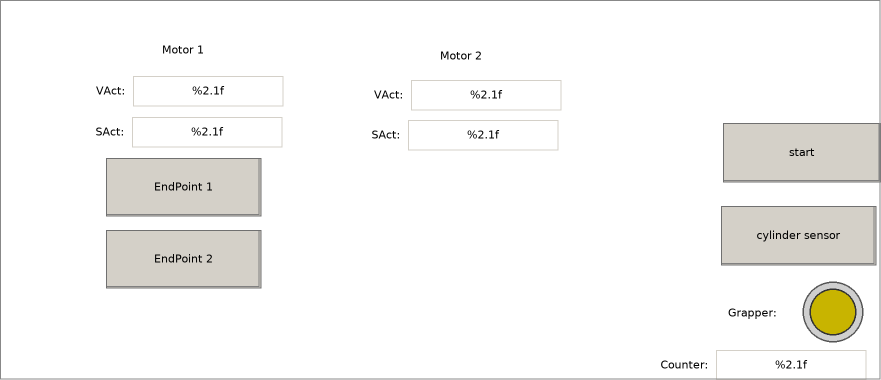
VISUALIZATION Visualization  // 881x380
    Button (723,123 158x59), "start"
        toggle GVL.StartStop
    Button (721,206 155x59), "cylinder sensor"
        toggle IO.A1_DI1
    Button (106,158 155x58), "EndPoint 1"
        tap IO.A1_DI2
    Button (106,230 155x58), "EndPoint 2"
        tap IO.A1_DI3
    Label (108,35 150x30), "Motor 1"
    Group (83,76 200x30)
        Label (0,0 45x30), "VAct:"
        Textfield (50,0 150x30), "%2.1f", text variable: GVL.motor1.VAct
    Group (84,117 198x30)
        Label (0,0 43x30), "SAct:"
        Textfield (48,0 150x30), "%2.1f", text variable: GVL.motor1.SAct
    Label (386,41 150x30), "Motor 2"
    Group (362,80 199x30)
        Label (0,0 44x30), "VAct:"
        Textfield (49,0 150x30), "%2.1f", text variable: GVL.motor2.VAct
    Group (365,120 193x30)
        Label (0,0 38x30), "SAct:"
        Textfield (43,0 150x30), "%2.1f", text variable: GVL.motor2.SAct
    Label (679,298 150x30), "Grapper:"
    Lamp1 (798,277 70x70), variable: A0_DO3, style: Lamp-Lamp1-Yellow
    Label (583,350 128x30), "Counter:"
    Textfield (716,350 150x30), "%2.1f", text variable: automat_PRG.counter
END_VISUALIZATION

(* stored: Version 1.1.0.1, ProductVersion 3.1.4024.12
   Visu Visualization: Id {f636cb6a-c664-44f8-be0c-b0b578fa4b1f} *)
